(* IEC 61131-3 sources: AXOpen/src/components.pneumatics/app/src, 2 files *)

(* ---- configuration.st ---- *)
USING AXOpen.Components.Pneumatics;

CONFIGURATION MyConfiguration
    TASK Main(Interval := T#1000ms, Priority := 1);
    PROGRAM P1 WITH Main: MyProgram;

    VAR_GLOBAL
        {S7.extern=ReadWrite}
        sandbox : SandboContext;
        {S7.extern=ReadWrite}
        documentation : DocumentationContext;
        {S7.extern=ReadWrite}
        _rtc : AXOpen.S71500.Rtc;
        {S7.extern=ReadWrite}
        _rtm : AXOpen.S71500.Rtm;
            {S7.extern=ReadWrite}
		HwInputs AT %IB0 : HwInputs;
        {S7.extern=ReadWrite}
		HwOutputs AT %QB0 : HwOutputs;
        {S7.extern=ReadWrite}
		PlcInputs : PlcInputs;
        {S7.extern=ReadWrite}
		PlcOutputs : PlcOutputs;
	END_VAR
END_CONFIGURATION

(* ---- program.st ---- *)
USING AXOpen.Components.Pneumatics;

PROGRAM MyProgram
    VAR_EXTERNAL
        sandbox : SandboxContext;
        documentation : DocumentationContext;
        _rtc : AXOpen.S71500.Rtc;
        _rtm : AXOpen.S71500.Rtm;
        PlcInputs : PlcInputs;
		PlcOutputs : PlcOutputs;
    END_VAR

    VAR

    END_VAR

    VAR_TEMP

    END_VAR
    CopyInputs();

    sandbox.PlcInputs := REF(PlcInputs);
    sandbox.PlcOutputs := REF(PlcOutputs);
    sandbox.Run();
    sandbox.InjectRtc(_rtc);
    sandbox.InjectRtm(_rtm);

    documentation.PlcInputs := REF(PlcInputs);
    documentation.PlcOutputs := REF(PlcOutputs);
    documentation.Run();
    documentation.InjectRtc(_rtc);
    documentation.InjectRtm(_rtm);

    CopyOutputs();
END_PROGRAM
